TYPE ST_AdsError EXTENDS ST_Error:
STRUCT
	Code	: TcError.AdsErrorCodes;
	Message	: Tc2_System.T_MaxString;
END_STRUCT
END_TYPE

(* stored: Version 1.1.0.1, ProductVersion 3.1.4024.14
   DUT ST_AdsError: Id {ccf3b3d3-ff0f-0d4f-2af5-045a6fb01ffd} *)
